TYPE (* logiBUS_DI Struct *)
  (* Version 1.0, 2025-07-21, franz *)
  PKP_2200_LI_DI_S : STRUCT
    Pin : USINT := 255;
  END_STRUCT;
END_TYPE
